FUNCTION FiniteStateMachine : E_FsmState
VAR_INPUT
	eArgFsmState : E_FsmState;
END_VAR
VAR
END_VAR

CASE eArgFsmState OF
	//0
	E_FsmState.ERR:
		FiniteStateMachine := E_FsmState.ERR;
	//1
	E_FsmState.INIT:
		FiniteStateMachine := E_FsmState.INIT;
	//2
	E_FsmState.STAT:
		FiniteStateMachine := E_FsmState.STAT;
	//3
	E_FsmState.STAT_TR:
		FiniteStateMachine := E_FsmState.STAT_TR;
	//4
	E_FsmState.NOM_LEV:
		FiniteStateMachine := E_FsmState.NOM_LEV;
	//5
	E_FsmState.INTER_TR:
		FiniteStateMachine := E_FsmState.INTER_TR;
	//6
	E_FsmState.END_TR:
		FiniteStateMachine := E_FsmState.END_TR;
END_CASE

END_FUNCTION

(* stored: Version 1.1.0.1, ProductVersion 3.1.4024.12
   POU FiniteStateMachine: Id {4331639f-1a7c-49f8-8301-e103bb836d39}, SpecialFunc None *)
